(* Logix 5000 project; controller Reto1 vendor 1 type 14 code 156 rev 30.11; software revision 30.00 *)

TASK MainTask (continuous, watchdog 500 ms) : MainProgram

MODULES
   Local : vendor 1 type 14 code 156 (Compact 0, rev 30.11)
      I_O : 1769-MODULE (Compact 3, rev 1.1, Output RPI 20 ms)
END_MODULES

VAR_GLOBAL   (* controller tags *)
   GD_IN_0 : BOOL;   // Sensor 1
   GD_IN_1 : BOOL;   // Sensor 2
   GD_IN_2 : BOOL;   // Sensor 3
   GD_IN_3 : BOOL;   // START GD
   GD_IN_4 : BOOL;   // Reset
   GD_IN_5 : BOOL;   // STOP GD
   GD_IN_6 : BOOL;   // STOP EMERGENCY GD
   GD_OUT_0 : BOOL;   // Barrera
   GD_OUT_5 : BOOL;   // Banda 2
END_VAR

PROGRAM MainProgram   (* main routine MainRoutine *)
VAR
   CajaLlego2 : BOOL;
   CajaPaso2 : BOOL;
   CajaPaso3 : BOOL;
   CondicionInicial : BOOL;
   ControlBarrera : BOOL;
   CounterCajas : COUNTER := (PRE := 1);
   Sensor2Down : BOOL;
   Sensor2Up : BOOL;
   Sensor3Up : BOOL;
   SistemaActivo : BOOL;
   TimerBarrera : TIMER := (PRE := 500);
END_VAR

ROUTINE MainRoutine   (* ladder *)
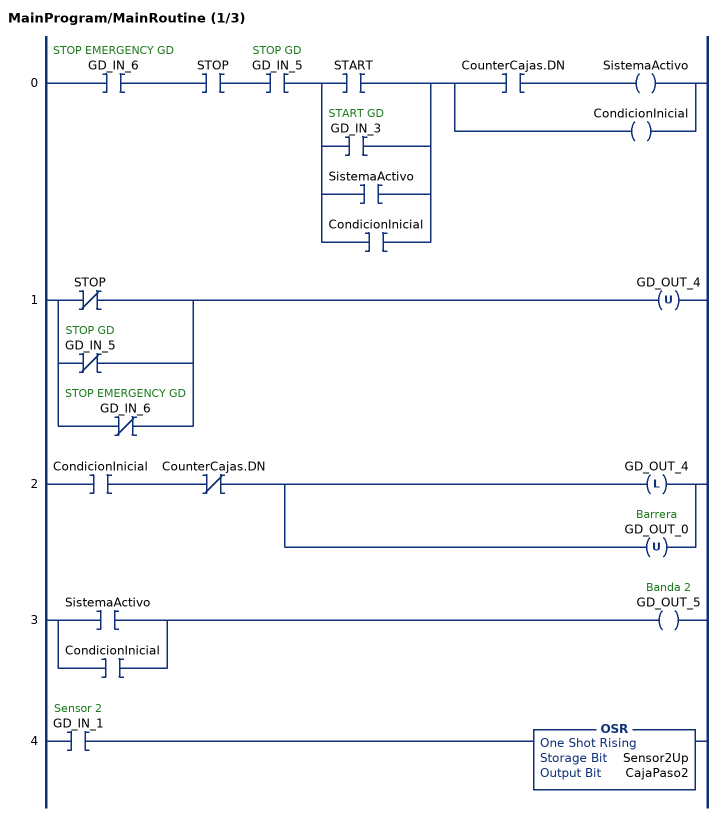
   0: XIC(GD_IN_6)XIC(STOP)XIC(GD_IN_5)[[XIC(START) ,XIC(GD_IN_3) ] ,[XIC(SistemaActivo) ,XIC(CondicionInicial) ] ][XIC(CounterCajas.DN) OTE(SistemaActivo) ,OTE(CondicionInicial) ];
   1: [XIO(STOP) ,[XIO(GD_IN_5) ,XIO(GD_IN_6) ] ]OTU(GD_OUT_4);
   2: XIC(CondicionInicial)XIO(CounterCajas.DN)[OTL(GD_OUT_4) ,OTU(GD_OUT_0) ];
   3: [XIC(SistemaActivo) ,XIC(CondicionInicial) ]OTE(GD_OUT_5);
   4: XIC(GD_IN_1)OSR(Sensor2Up,CajaPaso2);
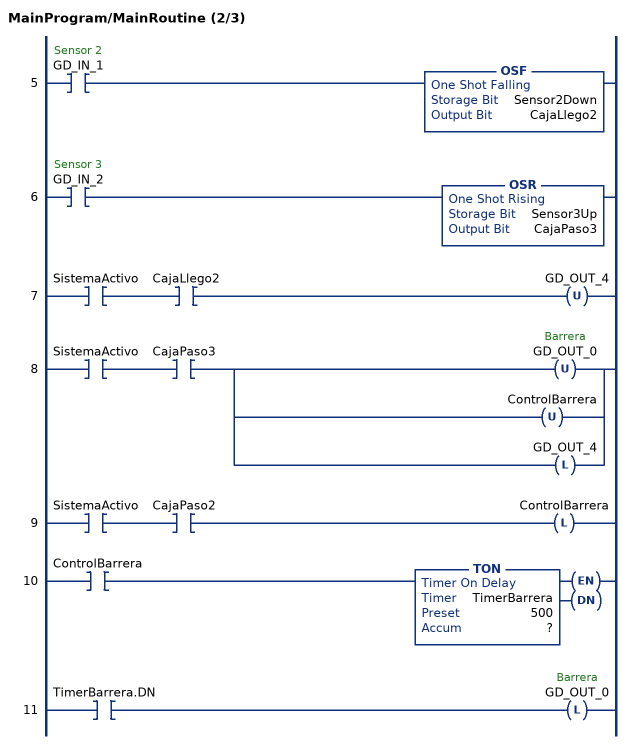
   5: XIC(GD_IN_1)OSF(Sensor2Down,CajaLlego2);
   6: XIC(GD_IN_2)OSR(Sensor3Up,CajaPaso3);
   7: XIC(SistemaActivo)XIC(CajaLlego2)OTU(GD_OUT_4);
   8: XIC(SistemaActivo)XIC(CajaPaso3)[OTU(GD_OUT_0) ,[OTU(ControlBarrera) ,OTL(GD_OUT_4) ] ];
   9: XIC(SistemaActivo)XIC(CajaPaso2)OTL(ControlBarrera);
   10: XIC(ControlBarrera)TON(TimerBarrera,?,?);
   11: XIC(TimerBarrera.DN)OTL(GD_OUT_0);
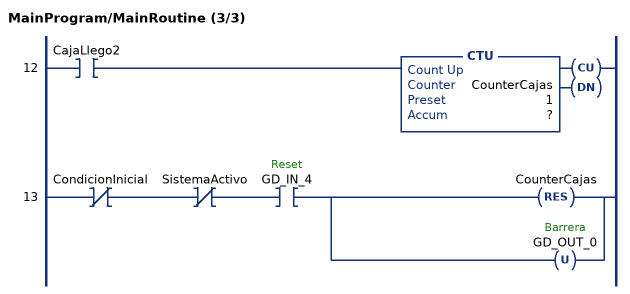
   12: XIC(CajaLlego2)CTU(CounterCajas,?,?);
   13: XIO(CondicionInicial)XIO(SistemaActivo)XIC(GD_IN_4)[RES(CounterCajas) ,OTU(GD_OUT_0) ];
END_ROUTINE
END_PROGRAM
